Staubli VAL3: setDryRunSig.pgx

public program setDryRunSig(bool enable_)
begin
  if enable_
    call debug:warning(libPath(),"Dry run mode enabled")
    dioLink(SYS:diEjcIn,SYS:doEjcIn)
    dioLink(SYS:diEjcOut,SYS:doEjcOut)
    dioLink(SYS:diCore1Pos1,SYS:doCore1Pos1)
    dioLink(SYS:diCore1Pos2,SYS:doCore1Pos2)
    dioLink(SYS:diCore2Pos1,SYS:doCore2Pos1)
    dioLink(SYS:diCore2Pos2,SYS:doCore2Pos2)
  else
    call debug:warning(libPath(),"Dry run mode disabled")
    call SYS:InitSysIO()
  endIf
end
